Universal Robots PolyScope program: sequential_p2.urp

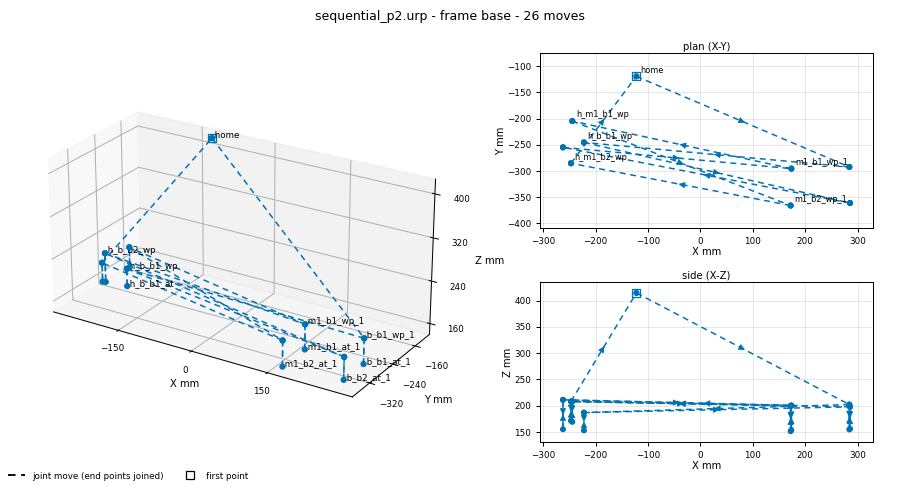
[picture p0: tool path of sequential_p2.urp in frame base, 26 of 26 moves have a stored position in this frame; points joined in program order, loops and branches not executed]
Program sequential_p2 (installation=default directory=/programs/ITER createdIn=5.3.1.64192 lastSavedIn=5.3.1.64192 robotSerialNumber=20195300365)
Calibrated DH parameters: a=[-0.000093, -0.190649, -0.212673, 0.000091, -0.000205, 0]; d=[0.151591, 44.061648, -42.488068, -1.442789, 0.085322, 0.091911]; alpha=[1.570082, -0.003447, 0.007513, 1.572293, -1.571904, 0]; deltaTheta=[0, -0.672656, 0.728185, -0.055522, 0.000005, 0]
Robot Program (runOnlyOnce=true)
  URCap Gripper Activate (Robotiq_Grippers, Robotiq Inc.) dataModel(ResetAndActivateKey=false)
  URCap Gripper (Robotiq_Grippers, Robotiq Inc.) dataModel(position=50.0, force=100.0, speed=100.0, positionInDouble=50.0, forceInDouble=100.0, speedInDouble=100.0, slaveIds=[9], blocking=true)
  MoveJ speed 60 deg/s, acceleration 80 deg/s^2 (useActiveTCP=true) feature=Base
    Waypoint home: TCP in base x=-122.15 y=-119.32 z=414.454 mm, rx=2.2563 ry=2.1459 rz=-0.0481 rad; joints [-85.681, -56.776, -79.802, -131.025, 89.944, -262.833] deg
  Folder Base
    MoveJ speed 60 deg/s, acceleration 80 deg/s^2 (useActiveTCP=true) feature=Base
      Waypoint b_b1_wp_1: TCP in base x=284.13 y=-292.134 z=202.324 mm, rx=2.2344 ry=2.1191 rz=-0.0341 rad; joints [-26.664, -114.085, -89.487, -63.473, 87.858, -203.352] deg
      Waypoint b_b1_at_1: TCP in base x=284.119 y=-292.135 z=154.941 mm, rx=2.2346 ry=2.1191 rz=-0.0343 rad; joints [-26.679, -119.503, -95.459, -52.092, 87.809, -203.308] deg
      URCap Gripper (Robotiq_Grippers, Robotiq Inc.) dataModel(position=100.0, force=100.0, speed=100.0, positionInDouble=100.0, forceInDouble=100.0, speedInDouble=100.0, slaveIds=[9], blocking=true)
      Waypoint b_b1_wp_2: TCP in base x=284.13 y=-292.134 z=202.324 mm, rx=2.2344 ry=2.1191 rz=-0.0341 rad; joints [-26.664, -114.085, -89.487, -63.473, 87.858, -203.352] deg
      Waypoint h_b_b1_wp: TCP in base x=-222.187 y=-245.349 z=187.06 mm, rx=-3.1315 ry=0.0204 rz=0.0123 rad; joints [-108.957, -99.116, -113.081, -58.146, 89.665, -197.782] deg
      Waypoint h_b_b1_at: TCP in base x=-222.188 y=-245.348 z=153.24 mm, rx=-3.1314 ry=0.0204 rz=0.0122 rad; joints [-108.969, -104.391, -117.643, -48.312, 89.612, -197.745] deg
      URCap Gripper (Robotiq_Grippers, Robotiq Inc.) dataModel(position=50.0, force=100.0, speed=100.0, positionInDouble=50.0, forceInDouble=100.0, speedInDouble=100.0, slaveIds=[9], blocking=true)
      Waypoint h_b_b1_wp: TCP in base x=-222.187 y=-245.349 z=187.06 mm, rx=-3.1315 ry=0.0204 rz=0.0123 rad; joints [-108.957, -99.116, -113.081, -58.146, 89.665, -197.782] deg
    MoveJ speed 60 deg/s, acceleration 80 deg/s^2 (useActiveTCP=true) feature=Base
      Waypoint b_b2_wp_1: TCP in base x=285.472 y=-360.969 z=198.014 mm, rx=2.2366 ry=2.1589 rz=-0.0532 rad; joints [-34.767, -127.303, -68.664, -72.529, 87.977, -212.535] deg
      Waypoint b_b2_at_1: TCP in base x=285.465 y=-360.98 z=156.253 mm, rx=2.2366 ry=2.1588 rz=-0.0532 rad; joints [-34.783, -130.917, -74.259, -63.319, 87.955, -212.495] deg
      URCap Gripper (Robotiq_Grippers, Robotiq Inc.) dataModel(position=100.0, force=100.0, speed=100.0, positionInDouble=100.0, forceInDouble=100.0, speedInDouble=100.0, slaveIds=[9], blocking=true)
      Waypoint b_b2_wp_2: TCP in base x=285.472 y=-360.969 z=198.014 mm, rx=2.2366 ry=2.1589 rz=-0.0532 rad; joints [-34.767, -127.303, -68.664, -72.529, 87.977, -212.535] deg
      Waypoint h_b_b2_wp: TCP in base x=-262.196 y=-254.726 z=211.351 mm, rx=-3.0605 ry=0.0443 rz=-0.0223 rad; joints [-114.749, -105.359, -96.042, -73.109, 89.199, -202.734] deg
      Waypoint h_b_b2_at: TCP in base x=-262.208 y=-254.718 z=155.33 mm, rx=-3.0605 ry=0.0443 rz=-0.0223 rad; joints [-114.774, -111.736, -104.192, -58.581, 89.146, -202.674] deg
      URCap Gripper (Robotiq_Grippers, Robotiq Inc.) dataModel(position=50.0, force=100.0, speed=100.0, positionInDouble=50.0, forceInDouble=100.0, speedInDouble=100.0, slaveIds=[9], blocking=true)
      Waypoint h_b_b2_wp: TCP in base x=-262.196 y=-254.726 z=211.351 mm, rx=-3.0605 ry=0.0443 rz=-0.0223 rad; joints [-114.749, -105.359, -96.042, -73.109, 89.199, -202.734] deg
  Folder Mid_1
    MoveJ speed 60 deg/s, acceleration 80 deg/s^2 (useActiveTCP=true) feature=Base
      Waypoint m1_b1_wp_1: TCP in base x=173.538 y=-295.326 z=200.585 mm, rx=2.2061 ry=2.2228 rz=-0.0106 rad; joints [-37.214, -100.014, -108.204, -61.217, 89.822, -217.247] deg
      Waypoint m1_b1_at_1: TCP in base x=173.554 y=-295.318 z=153.797 mm, rx=2.2061 ry=2.223 rz=-0.0106 rad; joints [-37.227, -106.714, -114.649, -48.075, 89.755, -217.198] deg
      URCap Gripper (Robotiq_Grippers, Robotiq Inc.) dataModel(position=100.0, force=100.0, speed=100.0, positionInDouble=100.0, forceInDouble=100.0, speedInDouble=100.0, slaveIds=[9], blocking=true)
      Waypoint m1_b1_wp_2: TCP in base x=173.538 y=-295.326 z=200.585 mm, rx=2.2061 ry=2.2228 rz=-0.0106 rad; joints [-37.214, -100.014, -108.204, -61.217, 89.822, -217.247] deg
      Waypoint h_m1_b1_wp: TCP in base x=-244.449 y=-204.582 z=208.1 mm, rx=2.2684 ry=2.1196 rz=0.0229 rad; joints [-116.825, -93.932, -112.747, -63.308, 92.582, -292.535] deg
      Waypoint h_m1_b1_at: TCP in base x=-244.447 y=-204.577 z=169.457 mm, rx=2.2685 ry=2.1196 rz=0.0229 rad; joints [-116.841, -99.299, -118.834, -51.852, 92.525, -292.487] deg
      URCap Gripper (Robotiq_Grippers, Robotiq Inc.) dataModel(position=50.0, force=100.0, speed=100.0, positionInDouble=50.0, forceInDouble=100.0, speedInDouble=100.0, slaveIds=[9], blocking=true)
      Waypoint h_m1_b1_wp: TCP in base x=-244.449 y=-204.582 z=208.1 mm, rx=2.2684 ry=2.1196 rz=0.0229 rad; joints [-116.825, -93.932, -112.747, -63.308, 92.582, -292.535] deg
    MoveJ speed 60 deg/s, acceleration 80 deg/s^2 (useActiveTCP=true) feature=Base
      Waypoint m1_b2_wp_1: TCP in base x=172.109 y=-365.692 z=199.867 mm, rx=2.2648 ry=2.1714 rz=0.0103 rad; joints [-46.162, -114.393, -88.528, -66.782, 90.646, -223.425] deg
      Waypoint m1_b2_at_1: TCP in base x=172.105 y=-365.689 z=151.683 mm, rx=2.2649 ry=2.1715 rz=0.0104 rad; joints [-46.178, -119.803, -94.665, -55.241, 90.602, -223.381] deg
      URCap Gripper (Robotiq_Grippers, Robotiq Inc.) dataModel(position=100.0, force=100.0, speed=100.0, positionInDouble=100.0, forceInDouble=100.0, speedInDouble=100.0, slaveIds=[9], blocking=true)
      Waypoint m1_b2_wp_2: TCP in base x=172.109 y=-365.692 z=199.867 mm, rx=2.2648 ry=2.1714 rz=0.0103 rad; joints [-46.162, -114.393, -88.528, -66.782, 90.646, -223.425] deg
      Waypoint h_m1_b2_wp: TCP in base x=-247.009 y=-285.144 z=208.116 mm, rx=2.2684 ry=2.1195 rz=0.0229 rad; joints [-111.389, -107.719, -95.772, -66.28, 92.556, -287.152] deg
      Waypoint h_m1_b2_at: TCP in base x=-246.994 y=-285.166 z=171.647 mm, rx=2.2684 ry=2.1196 rz=0.0229 rad; joints [-111.399, -111.783, -101.037, -56.949, 92.516, -287.113] deg
      URCap Gripper (Robotiq_Grippers, Robotiq Inc.) dataModel(position=50.0, force=100.0, speed=100.0, positionInDouble=50.0, forceInDouble=100.0, speedInDouble=100.0, slaveIds=[9], blocking=true)
      Waypoint h_m1_b2_wp: TCP in base x=-247.009 y=-285.144 z=208.116 mm, rx=2.2684 ry=2.1195 rz=0.0229 rad; joints [-111.389, -107.719, -95.772, -66.28, 92.556, -287.152] deg
  MoveJ speed 60 deg/s, acceleration 80 deg/s^2 (useActiveTCP=true) feature=Base
    Waypoint home: TCP in base x=-122.15 y=-119.32 z=414.454 mm, rx=2.2563 ry=2.1459 rz=-0.0481 rad; joints [-85.681, -56.776, -79.802, -131.025, 89.944, -262.833] deg
